FUNCTION_BLOCK T_Timer
VAR_INPUT
END_VAR
VAR
	task : T_Task;
	startTime : LINT; // ms
	_elapsedTimeInMs : LINT;
	_duration : LINT := 1;
	_signal : BOOL;
	_offSignal : BOOL;
END_VAR

{attribute 'monitoring' := 'call'} PROPERTY ElapsedTime : TIME
GET
ElapsedTime := LINT_TO_TIME( ElapsedTimeInMs );
END_GET
END_PROPERTY

{attribute 'monitoring' := 'call'} PROPERTY ElapsedTimeInMs : LINT
GET
ElapsedTimeInMs := task.DistributedClockTimeInMs - startTime;
END_GET
END_PROPERTY

PROPERTY Q_Off : BOOL
GET
Q_Off := _offSignal AND_THEN
			( ( task.DistributedClockTimeInMs - startTime ) > _duration );
END_GET
END_PROPERTY

PROPERTY Q_On : BOOL
GET
Q_On := _signal AND_THEN
			( ( task.DistributedClockTimeInMs - startTime ) > _duration );
END_GET
END_PROPERTY

PROPERTY Q_PulseTrain : BOOL
GET
Q_PulseTrain := _signal AND_THEN
			( ( task.DistributedClockTimeInMs - startTime ) MOD _duration > ( _duration / 2 ) );
END_GET
END_PROPERTY

PROPERTY SetPeriod : TIME
GET
SetPeriod := LINT_TO_TIME( _duration );
END_GET
SET
_duration := MAX( TIME_TO_LINT( SetPeriod ), 1);
END_SET
END_PROPERTY

PROPERTY Signal : BOOL
GET
Signal := _signal;
END_GET
SET
IF Signal <> _signal THEN
	startTime := task.DistributedClockTimeInMs;
	_signal := Signal;
	_offSignal := NOT _signal;
END_IF
END_SET
END_PROPERTY

END_FUNCTION_BLOCK

(* stored: Version 1.1.0.1, ProductVersion 3.1.4022.9
   POU T_Timer: Id {c856fe31-e123-4b16-a6bb-15d98c82e22c}, SpecialFunc None
   Property ElapsedTime: Id {8a9904e6-31e7-4e9d-b86a-65ffda125fec}
   Get Get: Id {488b6893-b0d4-43d1-9238-e2400fb8eeb8}
   Property ElapsedTimeInMs: Id {39ef3b5b-f7fe-40ca-8898-e880621dc8f1}
   Get Get: Id {d3f3f543-20a9-47bf-a9e3-ec99c7f0ed86}
   Property Q_Off: Id {08c2a48f-0dc0-49de-bf2d-183d52c59718}
   Get Get: Id {55ca00d5-a49d-4730-b3fd-217e8419398d}
   Property Q_On: Id {c1cc5243-5ef3-42dc-8554-e5a72de2db44}
   Get Get: Id {efe2eca9-3b6a-4325-8ce4-26b59119f648}
   Property Q_PulseTrain: Id {b920a6f9-c141-4439-bcab-162c60d1dcff}
   Get Get: Id {828a837c-2803-441e-a68b-cba172ccf9a3}
   Property SetPeriod: Id {33ba7951-e554-427e-81de-58f215094336}
   Get Get: Id {d87eca3d-708b-4edf-be46-377add0fce6b}
   Set Set: Id {bb954fa6-c7bf-4921-8824-f6432d76b967}
   Property Signal: Id {e88dd959-ce19-4a18-bb9b-dbb847f8258f}
   Get Get: Id {bec11fc9-db93-40f7-9738-dc0829db2d72}
   Set Set: Id {5d28a183-9130-4cf0-97a4-ce74854267a9} *)
